{attribute 'linkalways'} 
{attribute 'no_explicit_call' := 'This FB is a CLASS and must be accessed using methods or properties'}
{attribute 'enable_dynamic_creation'}
FUNCTION_BLOCK PUBLIC DeserializationFailedAlarm EXTENDS Alarm
VAR
	state : (CLEARED, RAISED);
	_reason : T_MAXSTRING;
END_VAR

PROPERTY Active : BOOL
GET
Active := state <> CLEARED;
END_GET
END_PROPERTY

METHOD PUBLIC Clear
_reason := '';
state := CLEARED;
END_METHOD

PROPERTY PUBLIC Message : T_MaxString
GET
Message := 'Deserialization failed';
END_GET
END_PROPERTY

METHOD PUBLIC Raise
VAR_INPUT
	Reason : T_MAXSTRING;
END_VAR
_reason := Reason;
state := RAISED;
END_METHOD

PROPERTY Reason : T_MaxString
GET
Reason := _reason;
END_GET
END_PROPERTY

END_FUNCTION_BLOCK

(* stored: Version 1.1.0.1, ProductVersion 3.1.4024.12
   POU DeserializationFailedAlarm: Id {20f48b43-fa78-4e08-b0ec-3b0d23aa70b0}, SpecialFunc None
   Property Active: Id {4057235a-9967-4e0b-b186-49a5b52f6495}
   Get Get: Id {5851e7d2-e662-4203-aa71-3ebaeba245e0}
   Method Clear: Id {26c4d86f-9f31-45ac-86e4-d0cdf5e647ea}
   Property Message: Id {0b3535dc-d696-4104-8384-6442be461f59}
   Get Get: Id {5368e9f4-f8a5-4bcb-a944-c8f6ed399cf1}
   Method Raise: Id {2493d769-8cd7-4765-85e9-6994872bd53d}
   Property Reason: Id {22470f33-ee70-4af3-ac4a-5e2470536b2e}
   Get Get: Id {1475eaa4-8066-4961-9a1f-f7525d2eb006} *)
